PROGRAM MAIN
VAR
END_VAR

END_PROGRAM

(* stored: Version 1.1.0.1, ProductVersion 3.1.4024.4
   POU MAIN: Id {29b549f1-d5e8-4154-b104-d1ebe480a748}, SpecialFunc None *)
